/// Specialized Config for SOR cell
TYPE ST_InputCellConfigurationGeneral :
STRUCT
	{attribute 'OPC.UA.DA.Description' := 'Dummy (for making struct visible on OPC UA'}
	Dummy						: BOOL;

END_STRUCT
END_TYPE

(* stored: Version 1.1.0.1, ProductVersion 3.1.4024.2
   DUT ST_InputCellConfigurationGeneral: Id {6a46902b-e007-46a9-b802-bc738795844d} *)
